(* IEC 61131-3 sources: UDPComm/src/Ar/UDPComm, 4 files *)

(* ---- UDPComm.typ ---- *)
(*
 * File: UDPComm.typ
 * Copyright (c) 2023 Loupe
 * https://loupe.team
 *
 * This file is part of UDPComm, licensed under the MIT License.
 *
 *)

TYPE

END_TYPE

(* ---- UDPCommMgr.typ ---- *)
(*
 * File: UDPCommMgr.typ
 * Copyright (c) 2023 Loupe
 * https://loupe.team
 *
 * This file is part of UDPComm, licensed under the MIT License.
 *
 *)

TYPE
	UDPCOMM_ERR_enum :
		(
		UDPCOMM_ERR_INVALIDINPUT := 50000,
		UDPCOMM_ERR_RECVDATATOOLARGE,
		UDPCOMM_ERR_SENDDATATOOLARGE,
		UDPCOMM_ERR_
		);
	UDPCOMM_ST_enum :
		(
		UDPCOMM_ST_CLOSED,
		UDPCOMM_ST_OPENING,
		UDPCOMM_ST_RUNNING,
		UDPCOMM_ST_CLOSING,
		UDPCOMM_ST_ERROR
		);
	UDPCOMM_SEND_ST_enum :
		(
		UDPCOMM_SEND_ST_IDLE,
		UDPCOMM_SEND_ST_SEND
		);
	UDPCommMgr_Int_FUB_typ : 	STRUCT
		Open : UdpOpen;
		Receive : UdpRecv;
		Send : UdpSend;
		Close : UdpClose;
	END_STRUCT;
	UDPCommMgr_Internal_typ : 	STRUCT
		CommState : UDPCOMM_ST_enum;
		ReceivedFromIPAddress : STRING[UDPCOMM_STRLEN_IPADDRESS];
		FUB : UDPCommMgr_Int_FUB_typ;
	END_STRUCT;
	UDPCommMgr_OUT_STAT_typ : 	STRUCT
		CommunicationActive : BOOL;
		Sending : BOOL;
		DataSent : BOOL;
		SentDataLength : UDINT;
		NewDataAvailable : BOOL;
		ReceivedDataLength : UDINT;
		ReceivedFromInterface : UDPCommMgr_Interface_typ;
		Ident : UDINT;
		Error : BOOL;
		ErrorID : UINT;
		ErrorString : STRING[UDPCOMM_STRLEN_ERRORSTRING];
	END_STRUCT;
	UDPCommMgr_OUT_typ : 	STRUCT
		STAT : UDPCommMgr_OUT_STAT_typ;
	END_STRUCT;
	UDPCommMgr_Interface_typ : 	STRUCT
		IPAddress : STRING[UDPCOMM_STRLEN_IPADDRESS] := 'IF1';
		Port : UINT;
	END_STRUCT;
	UDPCommMgr_IN_CFG_typ : 	STRUCT
		LocalInterface : UDPCommMgr_Interface_typ;
		RemoteInterface : UDPCommMgr_Interface_typ;
	END_STRUCT;
	UDPCommMgr_IN_PAR_typ : 	STRUCT
		AllowContinuousSend : BOOL;
		SendFlags : UINT;
		pSendData : UDINT;
		SendLength : UDINT;
		AllowContinuousReceive : BOOL;
		ReceiveFlags : UINT;
		pReceiveData : UDINT;
		MaxReceiveLength : UDINT;
		DisableReceiving : BOOL;
	END_STRUCT;
	UDPCommMgr_IN_CMD_typ : 	STRUCT
		Enable : BOOL;
		Send : BOOL;
		AcknowledgeData : BOOL;
		AcknowledgeError : BOOL;
	END_STRUCT;
	UDPCommMgr_IN_typ : 	STRUCT
		CMD : UDPCommMgr_IN_CMD_typ;
		PAR : UDPCommMgr_IN_PAR_typ;
		CFG : UDPCommMgr_IN_CFG_typ;
	END_STRUCT;
	UDPCommMgr_typ : 	STRUCT
		IN : UDPCommMgr_IN_typ;
		OUT : UDPCommMgr_OUT_typ;
		Internal : UDPCommMgr_Internal_typ;
	END_STRUCT;
END_TYPE

(* ---- UDPComm.fun ---- *)
(*
 * File: UDPComm.fun
 * Copyright (c) 2023 Loupe
 * https://loupe.team
 *
 * This file is part of UDPComm, licensed under the MIT License.
 *
 *)

FUNCTION UDPCommFn_Cyclic : UINT (*Cyclic function for managing UDP communications*) (*$GROUP=User*)
	VAR_IN_OUT
		t : UDPCommMgr_typ;
	END_VAR
END_FUNCTION

FUNCTION UDPCommManage : UINT (*Open and close UDP communication on the local interface*) (*$GROUP=User*)
	VAR_IN_OUT
		t : UDPCommMgr_typ;
	END_VAR
END_FUNCTION

FUNCTION UDPCommReceive : UINT (*Receive UDP datagrams*) (*$GROUP=User*)
	VAR_IN_OUT
		t : UDPCommMgr_typ;
	END_VAR
END_FUNCTION

FUNCTION UDPCommSend : UINT (*Send UDP datagrams*) (*$GROUP=User*)
	VAR_IN_OUT
		t : UDPCommMgr_typ;
	END_VAR
END_FUNCTION

(* ---- UDPComm.var ---- *)
(*
 * File: UDPComm.var
 * Copyright (c) 2023 Loupe
 * https://loupe.team
 *
 * This file is part of UDPComm, licensed under the MIT License.
 *
 *)
VAR CONSTANT
	UDPCOMM_MAI_DATA : UINT := 255;
	UDPCOMM_STRLEN_IPADDRESS : USINT := 16;
	UDPCOMM_STRLEN_ERRORSTRING : USINT := 80;
END_VAR
